FUNCTION_BLOCK MECHC_HMIL (* HMI for testing MECHC_VIEWL *)
  (* Standard: 61499-1; Classification: HMI; ApplicationDomain: SImulation *)
  (* Version 0.4, 2006-03-19, JHC, Holobloc Inc, Changed import to fb.rt.hmi *)
  (* Version 0.3, 2005-06-01, JHC, Holobloc Inc, Recompiled with new emitter. *)
  (* Version 0.2, 2004-09-27, JHC, Rockwell Automation, Changed order of variables for consistency with MECH_HMIL. *)
  (* Version 0.1, 2004-09-04, JHC, Rockwell Automation, Added FGD,BKGD. *)
  (* Version 0.0, 2002-05-21, JHC, Rockwell Automation, Copied/Modified from MECH_HMIL. *)
  (* Compiler header: package fb.rt.mva; import fb.rt.hmi.*; import fb.rt.net.*; *)
  (* Compiler classdef: public class MECHC_HMIL extends FBMVCD *)
  (* Compiler Java IBM VisualAge 3.0 *)
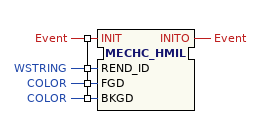
  EVENT_INPUT
    INIT WITH REND_ID, FGD, BKGD; (* Initialization Request *)
  END_EVENT
  EVENT_OUTPUT
    INITO; (* Initialization Confirm *)
  END_EVENT
  VAR_INPUT
    REND_ID : WSTRING; (* Data Channel ID - default is FB instaqnce name *)
    FGD : COLOR := red; (* Slider Foreground Color *)
    BKGD : COLOR := blue; (* Slider Background Color *)
  END_VAR
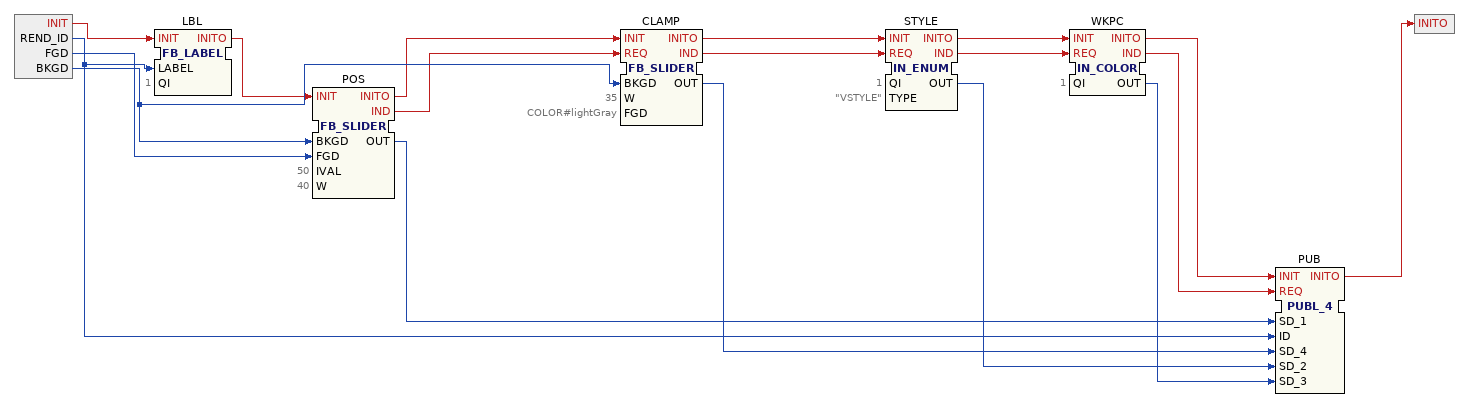
  FBS
    LBL : FB_LABEL(QI := 1);
    POS : FB_SLIDER(IVAL := 50, W := 40);
    CLAMP : FB_SLIDER(W := 35, FGD := COLOR#lightGray);
    STYLE : IN_ENUM(QI := 1, TYPE := "VSTYLE");
    WKPC : IN_COLOR(QI := 1);
    PUB : PUBL_4;
  END_FBS
  EVENT_CONNECTIONS
    INIT TO LBL.INIT;
    LBL.INITO TO POS.INIT;
    POS.INITO TO CLAMP.INIT;
    CLAMP.INITO TO STYLE.INIT;
    STYLE.INITO TO WKPC.INIT;
    WKPC.INITO TO PUB.INIT;
    PUB.INITO TO INITO;
    POS.IND TO CLAMP.REQ;
    CLAMP.IND TO STYLE.REQ;
    STYLE.IND TO WKPC.REQ;
    WKPC.IND TO PUB.REQ;
  END_CONNECTIONS
  DATA_CONNECTIONS
    POS.OUT TO PUB.SD_1;
    BKGD TO POS.BKGD;
    FGD TO POS.FGD;
    BKGD TO CLAMP.BKGD;
    REND_ID TO PUB.ID;
    REND_ID TO LBL.LABEL;
    CLAMP.OUT TO PUB.SD_4;
    STYLE.OUT TO PUB.SD_2;
    WKPC.OUT TO PUB.SD_3;
  END_CONNECTIONS
END_FUNCTION_BLOCK
